{attribute 'linkalways'} 
{attribute 'no_explicit_call' := 'This FB is a CLASS and must be accessed using methods or properties'}
{attribute 'enable_dynamic_creation'}
FUNCTION_BLOCK UnknownEnumerationError EXTENDS Error
VAR
	enumString : T_MAXSTRING;
END_VAR

PROPERTY PUBLIC ErrorType : T_MAXSTRING
GET
ErrorType := 'UNKNOWN_ENUMERATION_ERROR';
END_GET
END_PROPERTY

METHOD FB_init : BOOL
VAR_INPUT
	bInitRetains : BOOL; // if TRUE, the retain variables are initialized (warm start / cold start)
	bInCopyCode : BOOL;  // if TRUE, the instance afterwards gets moved into the copy code (online change)
	EnumString : T_MAXSTRING;
END_VAR
THIS^.enumString := EnumString;
END_METHOD

PROPERTY PUBLIC Message : T_MAXSTRING
GET
Message := CONCAT('Unknown Enumeration : ', enumString);
END_GET
END_PROPERTY

END_FUNCTION_BLOCK

(* stored: Version 1.1.0.1, ProductVersion 3.1.4024.12
   POU UnknownEnumerationError: Id {b1e0723b-943a-0c33-27eb-cdb4f968b150}, SpecialFunc None
   Folder Constructor: Id {704fc361-3a95-0555-39a6-d8f4052621ab}
   Property ErrorType: Id {05aa2827-c879-0b59-0e38-b997171f6124}
   Get Get: Id {1d6517f8-befc-05c7-3da9-b21ab4a4a9ed}
   Method FB_init: Id {60a21a1e-2b41-01d3-31c9-25219286f306}
   Property Message: Id {9aa7c44d-f725-0fd7-2562-1ef391f42ee3}
   Get Get: Id {dd97ac7c-9586-08eb-00e7-e9852e823684} *)
